(* IEC 61131-3 sources: programs/VI-54/VI-54_20171205/VI-54_20171205/Stations/PLC_VI54/VI-54_171014/Class/AlarmSleegersPara, 1 file *)

(* ---- AlarmSleegersPara.st ---- *)
(*!
<Class
	Name               = "AlarmSleegersPara"
	Revision           = "0.0"
	RealtimeTask       = "false"
	CyclicTask         = "false"
	BackgroundTask     = "false"
	Sigmatek           = "false"
	OSInterface        = "false"
	HighPriority       = "false"
	Automatic          = "false"
	UpdateMode         = "Prescan"
	SharedCommandTable = "true"
	Objectsize         = "(540,240)">
	<Channels>
		<Client Name="NextClass" Required="false" Internal="false"/>
	</Channels>
	<Network Name="AlarmSleegersPara">
		<!-- List of Components in this network -->
		<Components>
			<Object
				Name       = "_base"
				Class      = "_AlarmX0Para"
				Position   = "(218,120)"
				Visualized = "true"
				Remotely   = "true">
				<Channels>
					<Server Name="ClassSvr"/>
					<Client Name="Acknow"/>
					<Client Name="Config" Value="0"/>
					<Client Name="Group"/>
				</Channels>
			</Object>
		</Components>
		<Comments>
		</Comments>
		<!-- List of Connections in this network -->
		<Connections>
			<Connection Source="this.ClassSvr" Destination="_base.ClassSvr" Vertices="(690,210),(518,210),"/>
			<Connection Source="_base.Config" Destination="this.Config" Vertices="(218,210),(38,210),"/>
			<Connection Source="_base.Acknow" Destination="this.Acknow" Vertices="(218,270),(38,270),"/>
			<Connection Source="_base.Group" Destination="this.Group" Vertices="(218,330),(38,330),"/>
		</Connections>
		<!-- Headerfiles -->
		<Options>
		</Options>
	</Network>
</Class>
*)
#pragma using _AlarmX0Para

AlarmSleegersPara : CLASS
: _AlarmX0Para
  //Servers:
  //Clients:
	NextClass 	: CltChCmd_AlarmSleegersPara;
  //Variables:
		MachineNbr 	: DINT;
  //Functions:

	FUNCTION GLOBAL MyInit
		VAR_INPUT
			iStationNbr 	: DINT;
			iMachineNbr 	: DINT;
		END_VAR;

	FUNCTION GLOBAL AlarmState
		VAR_INPUT
			AlarmStr 	: tAlarm;
		END_VAR;
  //Tables:
	FUNCTION @STD
		VAR_OUTPUT
			ret_code	: CONFSTATES;
		END_VAR;
	FUNCTION GLOBAL TAB @CT_;
END_CLASS;

FUNCTION GLOBAL AlarmSleegersPara::MyInit
	VAR_INPUT
		iStationNbr 	: DINT;
		iMachineNbr 	: DINT;
	END_VAR

  // Set station number
  Config := (MachineNbr + iStationNbr);
  MachineNbr := iMachineNbr;

  if IsClientConnected(#NextClass) then
    NextClass.MyInit(iStationNbr:= (iStationNbr + 1), iMachineNbr:= MachineNbr);
  end_if;

END_FUNCTION

FUNCTION GLOBAL AlarmSleegersPara::AlarmState
	VAR_INPUT
		AlarmStr 	: tAlarm;
	END_VAR

  ClassSvr.Write(input:= AlarmStr[(Config - MachineNbr)]);

  if IsClientConnected(#NextClass) then
    NextClass.AlarmState(AlarmStr:= AlarmStr);
  end_if;

END_FUNCTION
